PROGRAM prg_Thermostaatregeling
VAR
	Thermostaat			AT		%I*		:REAL;
	Potentiometer1		AT		%I*		:INT;
	Potentiometer2		AT		%I*		:INT;
	
	Temperatuur			AT		%Q*		:REAL;
	Verwarming			AT		%Q*		:BOOL; //Is een Lamp
	TijdsRegeling: FB_WeeklyTimeSwitch;
	Dag: BOOL;

    fbTime : FB_LocalSystemTime;
    currentDT : DATE_AND_TIME;
END_VAR

//JE MOET VANONDER DE TIJDEN VAN EN TOT WANNEER AANPASSEN ALS JE DIT PROGRAMMA NIET TUSSEN
// 8u30 en 18u00 test

//SYSTEEM TIJD EN DATUM VOOR DE TIJDSREGELING HIERONDER:
fbTime(bEnable := TRUE);              // één keer starten, daarna cyclisch laten lopen
currentDT := SYSTEMTIME_TO_DT(fbTime.systemTime);

//programma met echte potentiometers van 0-32767:
//Thermostaat := 10.0 + (INT_TO_REAL(Potentiometer1) * 20.0 / 32767.0);
//Temperatuur := -30.0 + (INT_TO_REAL(Potentiometer2) * 70.0 / 32767.0);

//IF (Temperatuur < (Thermostaat - 1.0)) AND Dag THEN
//	Verwarming:=TRUE;
//ELSIF (Temperatuur >= (Thermostaat + 1.0)) OR NOT(Dag) THEN
//	Verwarming:=FALSE;
//END_IF

//Programma met de potentiometers in de visualisatie (anders verschaald)
Thermostaat := Potentiometer1;  // waarde van 10..30°C uit de Visu
Temperatuur := Potentiometer2;  // waarde van -30..40°C uit de Visu

IF (Temperatuur < (Thermostaat - 1.0)) AND Dag THEN
    Verwarming := TRUE;
ELSIF (Temperatuur >= (Thermostaat + 1.0)) OR NOT(Dag) THEN
    Verwarming := FALSE;
END_IF

//FunctieBlok uit library om tijdsinstellingen van 
TijdsRegeling(
	bEnable:= TRUE, 
	tCurrentDateTime:= currentDT, //hier moet een systeem variabele zoals CURRENT_DT of SYSTEM_DATE_AND_TIME maar vind ik niet
	tSwitchOnTime:= TOD#08:30, 
	tSwitchOffTime:= TOD#18:00, 
	bSunday:= TRUE, 
	bMonday:= TRUE, 
	bTuesday:= TRUE, 
	bWednesday:= TRUE, 	
	bThursday:= TRUE, 
	bFriday:= TRUE, 
	bSaturday:= TRUE, 
	bOutput=> Dag);

END_PROGRAM

(* stored: Version 1.1.0.1, ProductVersion 3.1.4024.15
   POU prg_Thermostaatregeling: Id {59be5007-5181-49e5-aaa0-53b8d85b4a2b}, SpecialFunc None *)
